{attribute 'TcGenerated'}
// This function has been automatically generated from the project information.
VAR_GLOBAL CONSTANT
    {attribute 'const_non_replaced'}
    {attribute 'linkalways'}
    stLibVersion_LFE_ARBITER : ST_LibVersion := (iMajor := 3, iMinor := 2, iBuild := 0, iRevision := 0, sVersion := '3.2.0');
END_VAR

(* stored: Version 1.1.0.1, ProductVersion 3.1.4022.18
   GVL Global_Version: Id 74cb9041-7547-41cf-9807-2b3a851b154b *)
